TYPE _ST_BLANK_1_ :
STRUCT
END_STRUCT
END_TYPE

(* stored: Version 1.1.0.1, ProductVersion 3.1.4022.18
   DUT _ST_BLANK_1_: Id {07a4109b-6159-431a-bc5b-70714945c6d7} *)
